{attribute 'qualified_only'}
{attribute 'strict'}
TYPE E_DiscreteValvePosition :
(	
	noValidInformation := 0,
	moving := 1,
	closed := 2,
	open := 3
);
END_TYPE

(* stored: Version 1.1.0.1, ProductVersion 3.1.4024.10
   DUT E_DiscreteValvePosition: Id {dde8a09a-e579-47ab-809c-5f9f7f9873ea} *)
